FUNCTION_BLOCK FB_BaseObjectEmulation
(**************************************************************************************
 * 	Application		:	BoxControl Framework
 *	Revision		:	$Revision: 404529 $
 *	Revision date	:	$Date: 2018-04-23 08:21:38 +0200 (Mo., 23 Apr 2018) $
 *	Last changed by	:	$Author: b7bolm $
 *	URL				:	$URL: http://almscdc.swisslog.com/repo/SWPD/Development/BoxControlFramework/20_Release/trunk/01_Software/BCF/BCF/JumpStart/20_Product/11_Emu/10_Base/10_Lib/FB_BaseObjectEmulation.TcPOU $
 *
 *	Purpose			:	Base object emulation
 *
 * ------------------------------------------------------------------------------------
 *	Copyright Swisslog [IP AG], Switzerland. All rights reserved.
 * 
 * ------------------------------------------------------------------------------------
 *	
 * 	Revision History: 
 *
 * 	VERSION			DATE			INITIALS			DESCRIPTION
 *	0.1				01.01.2001		swl					Example
 *
 **************************************************************************************)
VAR
	fbDebugMsg		: FB_DebugMsg; // Debug instance
	DebugMsg		: T_MAXSTRING; // Debug msg
END_VAR

(**************************************************************************************************************
   Body never called!
***************************************************************************************************************)
;

METHOD M_ITC_ProcessMsg : BOOL
VAR_INPUT
	meChannelSrc		: E_MFCS_CHANNEL; // Number of the source 
	mMsgType			: INT; // Message type
	mpData				: PVOID; // Data  pointer 
	mLen				: UDINT; // Data length
END_VAR
(*
This method serves as dummy to fullfil interface requirements.

This is needed to keep independency between library product types.

This method should be overwriten in each Rootclass underneath.

*)
END_METHOD

END_FUNCTION_BLOCK

(* stored: Version 1.1.0.1, ProductVersion 3.1.4022.12
   POU FB_BaseObjectEmulation: Id {7e7e997b-2e0e-4990-9ad3-247e61b2b611}, SpecialFunc None
   Method M_ITC_ProcessMsg: Id {671e3118-b495-4c4a-9f53-f45f38b37252} *)
